(*********************************** G.D S.p.A. - Technical Department ***********************************
============= PROGRAM INFO ============
FOLDER:             TBD
MACHINES INVOLVED:  TBD 

============= DESCRIPTION =============
csp machine declaration

============= REVISIONS ===============
Date		Version	 	Author      	Description             
----------	-------		------------  	--------------------------------------------
2019/04/05 	0000.00	 	M.Grasso		Creation of the PRG

**********************************************************************************************************)
(*$R process_ref := prc; $*)
PROGRAM csp_transfer_accumulator_accU_topRailWidth
VAR
	
	prc:									process;
	prc_path:								STRING;
	
	axis:									axis;
	Slot92_drv:								coe_drive;
	
	
	
END_VAR

VAR CONSTANT
	MOTOR_MAX_VELOCITY_DEGPS:				LREAL := 9600;
	MOTOR_MAX_ACCELLERATION_DEGPS2:			LREAL := 4800;
	MOTOR_MAX_DECELLERATION_DEGPS2:			LREAL := 4800;
	MOTOR_MAX_JERK_DEGPS3:					LREAL := 100000000; 
	MOTOR_MAX_FOLLOWING_ERROR_DEG:			LREAL := 2;
END_VAR

_read_var_input();

_object_manager();

IF NOT objects_running()
THEN
	RETURN;	
END_IF

_read_process_image();

_mode_manager();

_set_runtime_properties();

(********************************* BODY *********************************)
(************************************************************************)

_handle_messages();

_write_output();

ACTION _handle_messages:
;
END_ACTION

ACTION _handle_process_test:
;
END_ACTION

ACTION _mode_manager:
IF process_mode_req_is_pending(prc)
THEN
    process_apply_mode_req_first_step(prc);
    CASE process_get_mode(prc) OF
        MODE_TO_ABSENT:
			;
        MODE_TO_INACTIVE:
			;
        MODE_TO_TEST:
			;
        MODE_TO_OPERATIONAL:
			;
    END_CASE
    process_apply_mode_req_second_step(prc);
END_IF
END_ACTION

ACTION _object_manager:
IF objects_initialization()
THEN
	sub_process_init(
		object_name								:= 'csp_transfer_accumulator_accU_topRailWidth.prc', 
		process									:= csp_transfer_accumulator_accU.prc, 
		CONVERSION_this							:= prc);
		
	prc_path 									:= process_get_path(prc);
	
	axis_init(
		object_name								:= CONCAT(prc_path, '_axis'), 
		axis_type								:= AXIS_TYPE_SERVO, 
		encoder_scaling_factor					:= G_SERVO_ENCODER_SCALING_FACTOR_DEGPINC,
		modulo									:= G_MODULO_360_DEG, 
		process									:= prc, 
		CONVERSION_this							:= axis);
		
	axis_init_absolute_encoder_preset(	
		position								:=	0,
		CONVERSION_this							:=	axis);

	axis_set_max_dynamic(
		reference_velocity						:=	MOTOR_MAX_VELOCITY_DEGPS,
		velocity								:=	MOTOR_MAX_VELOCITY_DEGPS,
		acceleration							:=	MOTOR_MAX_ACCELLERATION_DEGPS2,
		deceleration							:=	MOTOR_MAX_DECELLERATION_DEGPS2,
		jerk									:=	MOTOR_MAX_JERK_DEGPS3,
		following_error							:=	MOTOR_MAX_FOLLOWING_ERROR_DEG,
		CONVERSION_this							:=	axis);
		
	coe_drive_init(
		object_name 							:= CONCAT(prc_path, '_Slot92_drv'),
		device_name 							:= 'IO61600Slot92 (EL7211)',
		vendor 									:= DRIVE_BECKHOFF_EL72x1,
		mode 									:= COE_DRIVE_MODE_DRIVEN_BY_AXIS,
		ethercat_master							:= csp_main.cabinet_transfer_ethercat_master,
		process									:= prc,
		CONVERSION_this 						:= Slot92_drv);

	axis_add_coe_drive(
		coe_drive								:= Slot92_drv,
		CONVERSION_this							:= axis);
	
	axis_add_safety_integrated_series(
		safety_integrated_series := csp_transfer_main_safety_accUChange.sis,
		CONVERSION_this := axis);
		
	
END_IF

IF objects_running()
THEN
	process_cycle(prc);
	axis_cycle(axis);
	coe_drive_cycle(Slot92_drv);
END_IF
END_ACTION

ACTION _read_process_image:
;
END_ACTION

ACTION _read_var_input:
;
END_ACTION

ACTION _set_runtime_properties:
;
END_ACTION

ACTION _write_output:
;
END_ACTION

END_PROGRAM

(* stored: Version 1.1.0.1, ProductVersion 3.1.4024.3
   POU csp_transfer_accumulator_accU_topRailWidth: Id {61162a2a-b24d-471d-8a98-0d3d95df92b7}, SpecialFunc None
   Action _handle_messages: Id {2bf1041e-10e1-48be-9a2e-21db195b12dd}
   Action _handle_process_test: Id {c1ca6184-12a6-4111-aa0c-2d87f1a58d96}
   Action _mode_manager: Id {c6cd768d-86ce-4277-8ba4-c76f524779af}
   Action _object_manager: Id {7e9af90f-3301-49a7-904a-3fb9749fdd41}
   Action _read_process_image: Id {bd6802e4-0c2d-4605-a946-05d702fae7e5}
   Action _read_var_input: Id {d2343f90-4a1e-43cd-a074-7775e4adaaa5}
   Action _set_runtime_properties: Id {745571af-634e-42c2-a7d6-92623cd6378d}
   Action _write_output: Id {2c0cb581-a431-4cbd-89ea-4f6502cc1d38} *)
